FUNCTION_BLOCK FB_TP (* standard timer function block (pulse) *)
  PACKAGE iec61131::timers;
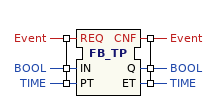
  EVENT_INPUT
    REQ WITH IN, PT; (* Service Request *)
  END_EVENT
  EVENT_OUTPUT
    CNF WITH Q, ET; (* Confirmation of Requested Service *)
  END_EVENT
  VAR_INPUT
    IN : BOOL; (* Input *)
    PT : TIME; (* Pulse time *)
  END_VAR
  VAR_OUTPUT
    Q : BOOL; (* output *)
    ET : TIME; (* elapse time *)
  END_VAR
  (* Service APPLICATION/RESOURCE: standard timer function block (pulse) *)
END_FUNCTION_BLOCK
